(* IEC 61131-3 sources: plc-example/, 3 files *)

(* ---- dut.iecst ---- *)
NAMESPACE MySpace
  TYPE ALARM : STRUCT
          State : BOOL; (* State of the alarm *)
          Confirmed : BOOL := FALSE; (* If confirmed *)
      END_STRUCT
  END_TYPE
END_NAMESPACE

(* ---- globals.iecst ---- *)
NAMESPACE GVL
    VAR_GLOBAL
        arAlarms : ARRAY[1..c_ALARMS_COUNT] OF MySpace.ALARM; (* List of alarms *)
    END_VAR

    VAR_GLOBAL CONSTANT
        c_ALARMS_COUNT : UINT := 10; (* Number of events *)
    END_VAR
END_NAMESPACE

(* ---- program.iecst ---- *)
PROGRAM PLC_PRG
   VAR
       xStart : BOOL; (* Comment *)
   END_VAR

   IF xStart = FALSE THEN
       GVL.arAlarms[1].state = TRUE;
   END_IF;

    METHOD init : BOOL
        xStart := TRUE;
    END_METHOD
END_PROGRAM
